{attribute 'analysis' := '-33'}
PROGRAM INTERNAL PRG_UnitTests
VAR
    {IF defined (UNIT_TEST)}
    fbParseRawInt32Tests    : 	FB_ParseRawInt32Tests;
    {END_IF}
END_VAR

{IF defined (UNIT_TEST)}

TcUnit.RUN();

{END_IF}

END_PROGRAM

(* stored: Version 1.1.0.1
   POU PRG_UnitTests: Id {c62e4430-fc3d-4856-ad8a-4ac6f6b51a31}, SpecialFunc None *)
